FUNCTION_BLOCK FB_Palletizer EXTENDS StateMachine
VAR_INPUT
END_VAR
VAR_OUTPUT
	
	bAllPartsPresent: BOOL;	
	
END_VAR
VAR
	fbPallBeltConveyor : FB_PalletizerConveyor;
	fbPallChainConveyor : FB_PalletizerConveyor;
	fbPallElevator : FB_PalletizerElevator;
	fbPushCyl : FB_Cylinder;
	fbTurnCyl : FB_Cylinder;
	fbPlateCyl : FB_Cylinder;
	fbClampCyl : FB_Cylinder;
	fbClampedSen : FB_Sensor;
	fbPlateLimitSen : FB_Sensor;
	fbPusherLimitSen : FB_Sensor;
	fbPresenceDetector : FB_PresenceDetector;
	fbDoneCycle : BoolOut;
	fbStepWorkerBusy : FB_StepWorker;
END_VAR

SUPER^();

fbPallBeltConveyor();
fbPallChainConveyor();
fbPushCyl();
fbTurnCyl();
fbPlateCyl();
fbClampCyl();
fbPresenceDetector(bAllPartsPresent => bAllPartsPresent);

METHOD PROTECTED   Busy : BOOL
VAR_INPUT
END_VAR
CASE fbStepWorkerBusy.uiStep OF

END_CASE
END_METHOD

METHOD PROTECTED  Error : BOOL
VAR_INPUT
END_VAR
END_METHOD

PROPERTY getDoneCycle : BoolOut
GET
getDoneCycle := fbDoneCycle;
END_GET
END_PROPERTY

METHOD PROTECTED  Init : BOOL
VAR_INPUT
END_VAR
Start();
END_METHOD

METHOD PROTECTED  Ready : BOOL
VAR_INPUT
END_VAR
END_METHOD

END_FUNCTION_BLOCK

(* stored: Version 1.1.0.1, ProductVersion 3.1.4024.0
   POU FB_Palletizer: Id {73a1f3d2-201c-42a5-94a2-081d42f8b358}, SpecialFunc None
   Method Busy: Id {d9e0814b-09a9-4c14-8872-e9e8a213db38}
   Method Error: Id {1e64e457-c3f7-4fa5-85b2-02fb48054177}
   Property getDoneCycle: Id {10630946-14f0-417b-8a72-9ea11d6f3ffa}
   Get Get: Id {81aca46c-aea3-436a-81f7-8d17ab991d2b}
   Method Init: Id {d70eb0e0-8e12-4f46-8c48-9d942d266afa}
   Method Ready: Id {42cd7ed1-7213-436f-b42d-812333345c3e} *)
